(* IEC 61131-3 sources: repolevel_ST_code_completion/output/0127完整版本_带planner/repoeval_three-axis_CNC_motion/readful_result_no_provide, 5 files *)

(* ---- FB_TripleAxisReset.st ---- *)
FUNCTION_BLOCK FB_TripleAxisReset
VAR_INPUT
<UNFIXABLE>
	bExecute		:	BOOL;				//执行复位信号
END_VAR
VAR_OUTPUT
	bDone			:	BOOL;				//三轴都复位完成
	bBusy			:	BOOL;				//复位进行中
	bError			:	BOOL;				//错误标志
	sErrorString	:	STRING;				//错误信息字符串
END_VAR
VAR
<UNFIXABLE>
	bResetXDone		:	BOOL;				//X轴复位完成标志
	bResetYDone		:	BOOL;				//Y轴复位完成标志
	bResetZDone		:	BOOL;				//Z轴复位完成标志
	bResetXError	:	BOOL;				//X轴复位错误标志
	bResetYError	:	BOOL;				//Y轴复位错误标志
	bResetZError	:	BOOL;				//Z轴复位错误标志
	sResetXError	:	STRING;				//X轴复位错误信息
	sResetYError	:	STRING;				//Y轴复位错误信息
	sResetZError	:	STRING;				//Z轴复位错误信息
END_VAR

IF NOT bExecute THEN
	bBusy := FALSE;
	bDone := FALSE;
	bError := FALSE;
	sErrorString := '';
	RETURN;
END_IF;

bBusy := TRUE;

// X轴复位
fbResetX(Execute := bExecute, Axis := AxisX);
bResetXDone := fbResetX.Done;
bResetXError := fbResetX.Error;
sResetXError := fbResetX.ErrorID;

// Y轴复位
fbResetY(Execute := bExecute, Axis := AxisY);
bResetYDone := fbResetY.Done;
bResetYError := fbResetY.Error;
sResetYError := fbResetY.ErrorID;

// Z轴复位
fbResetZ(Execute := bExecute, Axis := AxisZ);
bResetZDone := fbResetZ.Done;
bResetZError := fbResetZ.Error;
sResetZError := fbResetZ.ErrorID;

// 检查复位状态
IF bResetXError THEN
	bError := TRUE;
	sErrorString := CONCAT('X轴复位错误: ', sResetXError);
	bBusy := FALSE;
	RETURN;
END_IF;

IF bResetYError THEN
	bError := TRUE;
	sErrorString := CONCAT('Y轴复位错误: ', sResetYError);
	bBusy := FALSE;
	RETURN;
END_IF;

IF bResetZError THEN
	bError := TRUE;
	sErrorString := CONCAT('Z轴复位错误: ', sResetZError);
	bBusy := FALSE;
	RETURN;
END_IF;

IF bResetXDone AND bResetYDone AND bResetZDone THEN
	bDone := TRUE;
	bError := FALSE;
	sErrorString := '';
	bBusy := FALSE;
	RETURN;
END_IF;
END_FUNCTION_BLOCK

(* ---- FB_TripleAxisHoming.st ---- *)
VAR
	fbHomingX			:	SMC_HOMING;			//X轴回零功能块
	fbHomingY			:	SMC_HOMING;			//Y轴回零功能块
	fbHomingZ			:	SMC_HOMING;			//Z轴回零功能块
	bXHomingDone		:	BOOL;				//X轴回零完成标志
	bYHomingDone		:	BOOL;				//Y轴回零完成标志
	bZHomingDone		:	BOOL;				//Z轴回零完成标志
	bErrorDetected		:	BOOL;				//错误检测标志
	sLocalErrorString	:	STRING;				//本地错误信息
END_VAR

IF NOT bExecute THEN
	bBusy := FALSE;
	bHomeOK := FALSE;
	bAxisXHomeOK := FALSE;
	bAxisYHomeOK := FALSE;
	bAxisZHomeOK := FALSE;
	bError := FALSE;
	sErrorString := '';
	RETURN;
END_IF;

bBusy := TRUE;
bErrorDetected := FALSE;

// X轴回零逻辑
IF NOT bAxisXHomeOK THEN
	IF NOT bAxisXRefSwitch THEN
		fbHomingX.Axis := AxisX;
		fbHomingX.Velocity := fVelocityFast;
		fbHomingX.Acceleration := fAcceleration;
		fbHomingX.Deceleration := fDeceleration;
		fbHomingX.Execute := TRUE;
		IF fbHomingX.Error THEN
			bErrorDetected := TRUE;
			sLocalErrorString := 'X Axis Homing Error';
		END_IF;
	ELSE
		fbHomingX.Velocity := fVelocitySlow;
		IF fbHomingX.Done THEN
			bAxisXHomeOK := TRUE;
			fbHomingX.Execute := FALSE;
		END_IF;
	END_IF;
END_IF;

// Y轴回零逻辑
IF NOT bAxisYHomeOK AND NOT bErrorDetected THEN
	IF NOT bAxisYRefSwitch THEN
		fbHomingY.Axis := AxisY;
		fbHomingY.Velocity := fVelocityFast;
		fbHomingY.Acceleration := fAcceleration;
		fbHomingY.Deceleration := fDeceleration;
		fbHomingY.Execute := TRUE;
		IF fbHomingY.Error THEN
			bErrorDetected := TRUE;
			sLocalErrorString := 'Y Axis Homing Error';
		END_IF;
	ELSE
		fbHomingY.Velocity := fVelocitySlow;
		IF fbHomingY.Done THEN
			bAxisYHomeOK := TRUE;
			fbHomingY.Execute := FALSE;
		END_IF;
	END_IF;
END_IF;

// Z轴回零逻辑
IF NOT bAxisZHomeOK AND NOT bErrorDetected THEN
	IF NOT bAxisZRefSwitch THEN
		fbHomingZ.Axis := AxisZ;
		fbHomingZ.Velocity := fVelocityFast;
		fbHomingZ.Acceleration := fAcceleration;
		fbHomingZ.Deceleration := fDeceleration;
		fbHomingZ.Execute := TRUE;
		IF fbHomingZ.Error THEN
			bErrorDetected := TRUE;
			sLocalErrorString := 'Z Axis Homing Error';
		END_IF;
	ELSE
		fbHomingZ.Velocity := fVelocitySlow;
		IF fbHomingZ.Done THEN
			bAxisZHomeOK := TRUE;
			fbHomingZ.Execute := FALSE;
		END_IF;
	END_IF;
END_IF;

// 错误处理
IF bErrorDetected THEN
	bError := TRUE;
	sErrorString := sLocalErrorString;
	bBusy := FALSE;
	RETURN;
END_IF;

// 检查所有轴是否回零完成
IF bAxisXHomeOK AND bAxisYHomeOK AND bAxisZHomeOK THEN
	bHomeOK := TRUE;
	bBusy := FALSE;
END_IF;
END_FUNCTION_BLOCK

(* ---- FB_TripleAxisPower.st ---- *)
VAR
	fbPowerX		:	MC_POWER;			//X轴电源控制
	fbPowerY		:	MC_POWER;			//Y轴电源控制
	fbPowerZ		:	MC_POWER;			//Z轴电源控制
	bLocalError		:	BOOL;				//本地错误标志
	sLocalError		:	STRING;				//本地错误信息
END_VAR

IF NOT bServoEnable THEN
	bReady := FALSE;
	bAxisXReady := FALSE;
	bAxisYReady := FALSE;
	bAxisZReady := FALSE;
	bError := FALSE;
	sErrorString := '';
	RETURN;
END_IF;

// X轴电源控制
fbPowerX(
	Enable := bServoEnable,
	bRegulatorOn := bServoEnable,
	bDriveStart := bServoEnable,
	Axis := AxisX
);
bLocalError := fbPowerX.Error;
sLocalError := fbPowerX.ErrorID;

IF bLocalError THEN
	bError := TRUE;
	sErrorString := CONCAT('AxisX Error: ', sLocalError);
	bAxisXReady := FALSE;
ELSE
	bAxisXReady := fbPowerX.Status;
END_IF;

// Y轴电源控制
fbPowerY(
	Enable := bServoEnable,
	bRegulatorOn := bServoEnable,
	bDriveStart := bServoEnable,
	Axis := AxisY
);
bLocalError := fbPowerY.Error;
sLocalError := fbPowerY.ErrorID;

IF bLocalError THEN
	bError := TRUE;
	sErrorString := CONCAT('AxisY Error: ', sLocalError);
	bAxisYReady := FALSE;
ELSE
	bAxisYReady := fbPowerY.Status;
END_IF;

// Z轴电源控制
fbPowerZ(
	Enable := bServoEnable,
	bRegulatorOn := bServoEnable,
	bDriveStart := bServoEnable,
	Axis := AxisZ
);
bLocalError := fbPowerZ.Error;
sLocalError := fbPowerZ.ErrorID;

IF bLocalError THEN
	bError := TRUE;
	sErrorString := CONCAT('AxisZ Error: ', sLocalError);
	bAxisZReady := FALSE;
ELSE
	bAxisZReady := fbPowerZ.Status;
END_IF;

// 检查三轴是否都准备就绪
IF bAxisXReady AND bAxisYReady AND bAxisZReady THEN
	bReady := TRUE;
ELSE
	bReady := FALSE;
END_IF;
END_FUNCTION_BLOCK

(* ---- FB_TripleAxisStop.st ---- *)
VAR
	fbStopX			:	MC_STOP;			//X轴停止
	fbStopY			:	MC_STOP;			//Y轴停止
	fbStopZ			:	MC_STOP;			//Z轴停止
	bStopXDone		:	BOOL := FALSE;		//X轴停止完成标志
	bStopYDone		:	BOOL := FALSE;		//Y轴停止完成标志
	bStopZDone		:	BOOL := FALSE;		//Z轴停止完成标志
	bStopXError		:	BOOL := FALSE;		//X轴停止错误标志
	bStopYError		:	BOOL := FALSE;		//Y轴停止错误标志
	bStopZError		:	BOOL := FALSE;		//Z轴停止错误标志
	sStopXError		:	STRING := '';		//X轴错误信息
	sStopYError		:	STRING := '';		//Y轴错误信息
	sStopZError		:	STRING := '';		//Z轴错误信息
END_VAR

IF NOT bExecute THEN
	bDone := FALSE;
	bBusy := FALSE;
	RETURN;
END_IF;

bBusy := TRUE;
bDone := FALSE;
bError := FALSE;
sErrorString := '';

fbStopX(
	Execute := bExecute,
	Deceleration := rDeceleration,
	Axis := AxisX
);
bStopXDone := fbStopX.Done;
bStopXError := fbStopX.Error;
sStopXError := fbStopX.ErrorID;

fbStopY(
	Execute := bExecute,
	Deceleration := rDeceleration,
	Axis := AxisY
);
bStopYDone := fbStopY.Done;
bStopYError := fbStopY.Error;
sStopYError := fbStopY.ErrorID;

fbStopZ(
	Execute := bExecute,
	Deceleration := rDeceleration,
	Axis := AxisZ
);
bStopZDone := fbStopZ.Done;
bStopZError := fbStopZ.Error;
sStopZError := fbStopZ.ErrorID;

IF bStopXError THEN
	bError := TRUE;
	sErrorString := CONCAT('X轴错误: ', sStopXError);
	bBusy := FALSE;
	RETURN;
END_IF;

IF bStopYError THEN
	bError := TRUE;
	sErrorString := CONCAT('Y轴错误: ', sStopYError);
	bBusy := FALSE;
	RETURN;
END_IF;

IF bStopZError THEN
	bError := TRUE;
	sErrorString := CONCAT('Z轴错误: ', sStopZError);
	bBusy := FALSE;
	RETURN;
END_IF;

IF bStopXDone AND bStopYDone AND bStopZDone THEN
	bDone := TRUE;
	bBusy := FALSE;
	RETURN;
END_IF;
END_FUNCTION_BLOCK

(* ---- INIT_CNC_System.st ---- *)
fbSMC_ReadNCFile(bExecute := FALSE);
fbSMC_ReadNCFile(bExecute := TRUE);

fbSMC_NCDecoder(bExecute := FALSE, ncprog := fbSMC_ReadNCFile.ncprog);
fbSMC_NCDecoder(bExecute := TRUE, ncprog := fbSMC_ReadNCFile.ncprog);

fbSMC_CheckVelocities(bExecute := FALSE);
fbSMC_CheckVelocities(bExecute := TRUE);

fbSMC_Interpolator(bExecute := FALSE);
fbSMC_Interpolator(bExecute := TRUE);

fbSMC_ControlAxisXByPos(bExecute := FALSE, Axis := AxisX);
fbSMC_ControlAxisXByPos(bExecute := TRUE, Axis := AxisX);

fbSMC_ControlAxisYByPos(bExecute := FALSE, Axis := AxisY);
fbSMC_ControlAxisYByPos(bExecute := TRUE, Axis := AxisY);

fbSMC_ControlAxisZByPos(bExecute := FALSE, Axis := AxisZ);
fbSMC_ControlAxisZByPos(bExecute := TRUE, Axis := AxisZ);

fbSMC_AXISX_HOMING(bExecute := FALSE, Axis := AxisX);
fbSMC_AXISX_HOMING(bExecute := TRUE, Axis := AxisX);

fbSMC_AXISY_HOMING(bExecute := FALSE, Axis := AxisY);
fbSMC_AXISY_HOMING(bExecute := TRUE, Axis := AxisY);

fbSMC_AXISZ_HOMING(bExecute := FALSE, Axis := AxisZ);
fbSMC_AXISZ_HOMING(bExecute := TRUE, Axis := AxisZ);

fbMC_AXISX_STOP(bExecute := FALSE, Axis := AxisX);
fbMC_AXISX_STOP(bExecute := TRUE, Axis := AxisX);

fbMC_AXISY_STOP(bExecute := FALSE, Axis := AxisY);
fbMC_AXISY_STOP(bExecute := TRUE, Axis := AxisY);

fbMC_AXISZ_STOP(bExecute := FALSE, Axis := AxisZ);
fbMC_AXISZ_STOP(bExecute := TRUE, Axis := AxisZ);

RETURN := TRUE;
END_FUNCTION
